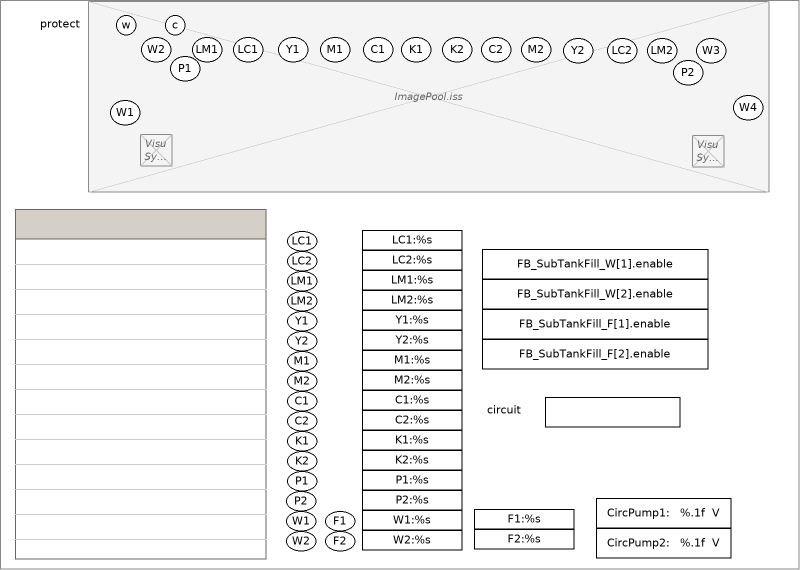
VISUALIZATION VIS_SubTank  // 800x570
    Image (88,1 681x191), image: ImagePool.iss
    Ellipse (116,15 20x20), "w", colour toggle: stInput.biProtectAirTankLevel_W
        toggle stInput.biProtectAirTankLevel_W
    Label (30,9 60x30), "protect"
    Ellipse (165,15 20x20), "c", colour toggle: stInput.biProtectAirTankLevel_C
        toggle stInput.biProtectAirTankLevel_C
    Group (110,37 653x130)
        Ellipse (0,63 30x25), "W1", colour toggle: stInput.biSubInkTankLevel[13]
            toggle stInput.biSubInkTankLevel[15]
        Ellipse (31,0 30x25), "W2", colour toggle: stInput.biSubInkTankLevel[14]
            toggle stInput.biSubInkTankLevel[16]
        Ellipse (123,0 30x25), "LC1", colour toggle: stInput.biSubInkTankLevel[1]
            toggle stInput.biSubInkTankLevel[11]
        Ellipse (82,0 30x25), "LM1", colour toggle: stInput.biSubInkTankLevel[3]
            toggle stInput.biSubInkTankLevel[9]
        Ellipse (168,0 30x25), "Y1", colour toggle: stInput.biSubInkTankLevel[5]
            toggle stInput.biSubInkTankLevel[1]
        Ellipse (210,0 30x25), "M1", colour toggle: stInput.biSubInkTankLevel[7]
            toggle stInput.biSubInkTankLevel[3]
        Ellipse (253,0 30x25), "C1", colour toggle: stInput.biSubInkTankLevel[9]
            toggle stInput.biSubInkTankLevel[5]
        Ellipse (291,0 30x25), "K1", colour toggle: stInput.biSubInkTankLevel[11]
            toggle stInput.biSubInkTankLevel[7]
        Ellipse (332,0 30x25), "K2", colour toggle: stInput.biSubInkTankLevel[12]
            toggle stInput.biSubInkTankLevel[8]
        Ellipse (371,0 30x25), "C2", colour toggle: stInput.biSubInkTankLevel[10]
            toggle stInput.biSubInkTankLevel[6]
        Ellipse (411,0 30x25), "M2", colour toggle: stInput.biSubInkTankLevel[8]
            toggle stInput.biSubInkTankLevel[4]
        Ellipse (453,1 30x25), "Y2", colour toggle: stInput.biSubInkTankLevel[6]
            toggle stInput.biSubInkTankLevel[2]
        Ellipse (537,1 30x25), "LM2", colour toggle: stInput.biSubInkTankLevel[4]
            toggle stInput.biSubInkTankLevel[10]
        Ellipse (497,1 30x25), "LC2", colour toggle: stInput.biSubInkTankLevel[2]
            toggle stInput.biSubInkTankLevel[12]
        Ellipse (586,1 30x25), "W3", colour toggle: stInput.biSubInkTankLevel[15]
            toggle stInput.biSubInkTankLevel[17]
        Ellipse (623,58 30x25), "W4", colour toggle: stInput.biSubInkTankLevel[16]
            toggle stInput.biSubInkTankLevel[18]
        Image (30,97 32x32), colour toggle: stOutput.bqSubCircPumpWorking[1], image: VisuSymbols.Symbols.ArrowQuarterLeftUp
        Image (582,98 32x32), colour toggle: stOutput.bqSubCircPumpWorking[2], image: VisuSymbols.Symbols.ArrowQuarterRightUp
        Ellipse (60,19 30x25), "P1", colour toggle: stInput.biSubInkTankLevel[17]
            toggle stInput.biSubInkTankLevel[13]
        Ellipse (563,23 30x25), "P2", colour toggle: stInput.biSubInkTankLevel[18]
            toggle stInput.biSubInkTankLevel[14]
    Ellipse (287,231 30x20), "LC1", colour toggle: stOutput.bqFillPumpWorking[1]
    Ellipse (287,271 30x20), "LM1", colour toggle: stOutput.bqFillPumpWorking[3]
    Ellipse (287,311 30x20), "Y1", colour toggle: stOutput.bqFillPumpWorking[5]
    Ellipse (287,351 30x20), "M1", colour toggle: stOutput.bqFillPumpWorking[7]
    Ellipse (287,391 30x20), "C1", colour toggle: stOutput.bqFillPumpWorking[9]
    Ellipse (287,251 30x20), "LC2", colour toggle: stOutput.bqFillPumpWorking[2]
    Ellipse (287,291 30x20), "LM2", colour toggle: stOutput.bqFillPumpWorking[4]
    Ellipse (287,331 30x20), "Y2", colour toggle: stOutput.bqFillPumpWorking[6]
    Ellipse (287,371 30x20), "M2", colour toggle: stOutput.bqFillPumpWorking[8]
    Ellipse (287,411 30x20), "C2", colour toggle: stOutput.bqFillPumpWorking[10]
    Ellipse (287,431 30x20), "K1", colour toggle: stOutput.bqFillPumpWorking[11]
    Ellipse (287,451 30x20), "K2", colour toggle: stOutput.bqFillPumpWorking[12]
    Ellipse (286,531 30x20), "W2", colour toggle: stOutput.bqFillPumpWorking[15]
    Ellipse (286,491 30x20), "P2", colour toggle: stOutput.bqFillPumpWorking[18]
    Ellipse (325,531 30x20), "F2", colour toggle: stOutput.bqFillPumpWorking[20]
    Ellipse (286,511 30x20), "W1", colour toggle: stOutput.bqFillPumpWorking[13]
    Ellipse (287,471 30x20), "P1", colour toggle: stOutput.bqFillPumpWorking[17]
    Ellipse (325,511 30x20), "F1", colour toggle: stOutput.bqFillPumpWorking[19]
    Rectangle (362,230 100x20), "LC1:%s", text variable: P_SubTank.FB_SubTankFill_C[1].inkFillTimeOutTon.ET
    Rectangle (362,270 100x20), "LM1:%s", text variable: P_SubTank.FB_SubTankFill_C[3].inkFillTimeOutTon.ET
    Rectangle (362,310 100x20), "Y1:%s", text variable: P_SubTank.FB_SubTankFill_C[5].inkFillTimeOutTon.ET
    Rectangle (362,350 100x20), "M1:%s", text variable: P_SubTank.FB_SubTankFill_C[7].inkFillTimeOutTon.ET
    Rectangle (362,390 100x20), "C1:%s", text variable: P_SubTank.FB_SubTankFill_C[9].inkFillTimeOutTon.ET
    Rectangle (362,430 100x20), "K1:%s", text variable: P_SubTank.FB_SubTankFill_C[11].inkFillTimeOutTon.ET
    Rectangle (362,510 100x20), "W1:%s", text variable: P_SubTank.FB_SubTankFill_W[1].inkFillTimeOutTon.ET
    Rectangle (362,470 100x20), "P1:%s", text variable: P_SubTank.FB_SubTankFill_P[1].inkFillTimeOutTon.ET
    Rectangle (474,509 100x20), "F1:%s", text variable: P_SubTank.FB_SubTankFill_F[1].inkFillTimeOutTon.ET
    Rectangle (362,250 100x20), "LC2:%s", text variable: P_SubTank.FB_SubTankFill_C[2].inkFillTimeOutTon.ET
    Rectangle (362,290 100x20), "LM2:%s", text variable: P_SubTank.FB_SubTankFill_C[4].inkFillTimeOutTon.ET
    Rectangle (362,330 100x20), "Y2:%s", text variable: P_SubTank.FB_SubTankFill_C[6].inkFillTimeOutTon.ET
    Rectangle (362,370 100x20), "M2:%s", text variable: P_SubTank.FB_SubTankFill_C[8].inkFillTimeOutTon.ET
    Rectangle (362,410 100x20), "C2:%s", text variable: P_SubTank.FB_SubTankFill_C[10].inkFillTimeOutTon.ET
    Rectangle (362,450 100x20), "K2:%s", text variable: P_SubTank.FB_SubTankFill_C[12].inkFillTimeOutTon.ET
    Rectangle (362,530 100x20), "W2:%s", text variable: P_SubTank.FB_SubTankFill_W[2].inkFillTimeOutTon.ET
    Rectangle (362,490 100x20), "P2:%s", text variable: P_SubTank.FB_SubTankFill_P[2].inkFillTimeOutTon.ET
    Rectangle (474,529 100x20), "F2:%s", text variable: P_SubTank.FB_SubTankFill_f[2].inkFillTimeOutTon.ET
    Rectangle (596,498 135x30), "CircPump1: %.1f V", text variable: HMI_CircPump1_V
        OnMouseDown: write HMI_CircPump1_V via Default, min 0, max 5
    Rectangle (596,528 135x30), "CircPump2: %.1f V", text variable: HMI_CircPump2_V
        OnMouseDown: write HMI_CircPump2_V via Default, min 0, max 5
    Rectangle (545,397 135x30), text list: 'TextList_SubTank_circuit', text index: SubTankInk_type
        OnMouseDown: write HMI_CircPump1_V via Default, min 0, max 5
    Rectangle (482,249 226x30), "FB_SubTankFill_W[1].enable", text variable: HMI_CircPump1_V, colour toggle: P_SubTank.FB_SubTankFill_W[1].enable
        OnMouseDown: write HMI_CircPump1_V via Default, min 0, max 5
    Rectangle (482,279 226x30), "FB_SubTankFill_W[2].enable", text variable: HMI_CircPump1_V, colour toggle: P_SubTank.FB_SubTankFill_W[2].enable
        OnMouseDown: write HMI_CircPump1_V via Default, min 0, max 5
    Rectangle (482,339 226x30), "FB_SubTankFill_F[2].enable", text variable: HMI_CircPump1_V, colour toggle: P_SubTank.FB_SubTankFill_F[2].enable
        OnMouseDown: write HMI_CircPump1_V via Default, min 0, max 5
    Rectangle (482,309 226x30), "FB_SubTankFill_F[1].enable", text variable: HMI_CircPump1_V, colour toggle: P_SubTank.FB_SubTankFill_F[1].enable
        OnMouseDown: write HMI_CircPump1_V via Default, min 0, max 5
    Label (474,395 60x30), "circuit"
    Table (15,209 251x350), data array: GVL_API.stSubTank
        p3854506369: GVL_API.stSubTank[INDEX].error_code
        p1892666644: GVL_API.stSubTank[INDEX].state
        p338671338: GVL_API.stSubTank[INDEX].Error
        p2170511999: GVL_API.stSubTank[INDEX].Setoff
        Columns.Column.[3].Template: toggle GVL_API.stSubTank[INDEX].Setoff
END_VISUALIZATION

(* stored: Version 1.1.0.1, ProductVersion 3.1.4024.11
   Visu VIS_SubTank: Id {672d6fbc-a79f-49be-9b61-cee8e7a1663c} *)
